Staubli VAL3: getObjectData.pgx

public program getObjectData(num x_nConvNum (dimensions=1), trsf& x_trObject[] (dimensions=1), num& x_nError[] (dimensions=1))
  local point l_pPoint
begin
  // This program returns the coordinates of the object
  // that have been pushed into the buffer by the detection lib
  // of the specified conveyor.
  // This function is usefull when an advanced detection device
  // (e.g vision system) is in use.
  //
  // Input Param
  //  x_nConvNum  : Conveyor number
  //
  // Output Param
  //  x_trObject  : coordinates of the object
  //  x_nError    : Error code
  //    0 : No error
  //    1 : No data available
  //
  //----------------------------------------------------------------
  //
  switch x_nConvNum
    case 0
      call cnv0:getObjectData(x_trObject,x_nError)
    break
    case 1
      call cnv1:getObjectData(x_trObject,x_nError)
    break
  endSwitch
end
